// TwinCAT 3 PLC project pruebaAlmacenje
// ProgramVersion: 3.1.4024.0
// libraries:
//   Tc2_Standard, * (Beckhoff Automation GmbH)
//   Tc2_System, * (Beckhoff Automation GmbH)
//   Tc3_Module, * (Beckhoff Automation GmbH)
// project tree:
//   GVLs/ GVLvar.TcGVL (not stored)
//   / PlcTask.TcTTO
//   POUs/ MAIN.TcPOU, posicionEstanteria.TcPOU (not stored), distanciaBaldas.TcPOU
// real-time tasks:
//   TASK PlcTask: cycle T#10ms, priority 20, ADS port 350

CONFIGURATION pruebaAlmacenje
    RESOURCE PLC ON TwinCAT3
        TASK PlcTask(INTERVAL := T#10ms, PRIORITY := 20);
        PROGRAM MAIN WITH PlcTask : MAIN;
    END_RESOURCE
END_CONFIGURATION

// ---- POUs/MAIN.TcPOU
PROGRAM MAIN
VAR
	enclaveStart: BOOL;
	timerColumna: TON;
	posicionEst : ARRAY[1..2] OF REAL;
	distBaldas : distanciaBaldas();
END_VAR

(*
clumnas 1.6 - 1
filas 0.5-2.1
*)


IF GVLvar.botonStart THEN
	enclaveStart := TRUE;
	GVLvar.cinta := TRUE;
	distBaldas();
END_IF


IF enclaveStart THEN
	
	//si hay una caja en la enrada apr almacenar se prepara la grua
	IF GVLvar.sensorEntradaGrua THEN
		GVLvar.cinta := FALSE;
		posicionEst := posicionEstanteria();
		GVLvar.setPointX := posicionEst[1];
		GVLvar.setPointZ := posicionEst[2];
		//flanco de bajada en la senal de movimiento
		// xq si no se para automaticamente la grua al apsar al else
	ELSE
		GVLvar.setPointX := 0.0;
		GVLvar.setPointZ := 0.0;
	END_IF
	
	
END_IF

END_PROGRAM

// ---- POUs/distanciaBaldas.TcPOU
FUNCTION_BLOCK distanciaBaldas
VAR_INPUT
END_VAR
VAR_OUTPUT
END_VAR
VAR
END_VAR

// Fila 1
GVLvar.estanteria[1,1][1] := 1.6;  GVLvar.estanteria[1,1][2] := 0.5;
GVLvar.estanteria[1,2][1] := 2.7;  GVLvar.estanteria[1,2][2] := 0.5;
GVLvar.estanteria[1,3][1] := 3.7;  GVLvar.estanteria[1,3][2] := 0.5;

// Fila 2
GVLvar.estanteria[2,1][1] := 1.6;  GVLvar.estanteria[2,1][2] := 2.1;
GVLvar.estanteria[2,2][1] := 2.7;  GVLvar.estanteria[2,2][2] := 2.1;
GVLvar.estanteria[2,3][1] := 3.7;  GVLvar.estanteria[2,3][2] := 2.1;

// Fila 3
GVLvar.estanteria[3,1][1] := 1.6;  GVLvar.estanteria[3,1][2] := 3.9;
GVLvar.estanteria[3,2][1] := 2.7;  GVLvar.estanteria[3,2][2] := 3.9;
GVLvar.estanteria[3,3][1] := 3.7;  GVLvar.estanteria[3,3][2] := 3.9;

// Fila 4
GVLvar.estanteria[4,1][1] := 1.6;  GVLvar.estanteria[4,1][2] := 5.6;
GVLvar.estanteria[4,2][1] := 2.7;  GVLvar.estanteria[4,2][2] := 5.6;
GVLvar.estanteria[4,3][1] := 3.7;  GVLvar.estanteria[4,3][2] := 5.6;

// Fila 5
GVLvar.estanteria[5,1][1] := 1.6;  GVLvar.estanteria[5,1][2] := 8.3;
GVLvar.estanteria[5,2][1] := 2.7;  GVLvar.estanteria[5,2][2] := 8.3;
GVLvar.estanteria[5,3][1] := 3.7;  GVLvar.estanteria[5,3][2] := 8.3;

// Fila 6
GVLvar.estanteria[6,1][1] := 1.6;  GVLvar.estanteria[6,1][2] := 8.7;
GVLvar.estanteria[6,2][1] := 2.7;  GVLvar.estanteria[6,2][2] := 8.7;
GVLvar.estanteria[6,3][1] := 3.7;  GVLvar.estanteria[6,3][2] := 8.7;

END_FUNCTION_BLOCK
